// SIMATIC S7-200 project (STEP 7-Micro/WIN), CPU 224XP REL 02.01

SYMBOL_TABLE USUARIO1
P_MOTOR1         I0.0
P_MOTOR2         I0.1
P_PARO           I0.2
MOTOR_1          Q0.0
MOTOR_2          Q0.1
COUNT_SG_M1      VW0      // VARIABLE ENCARGADA DE CONTAR LOS SG DE FUNCIONAMIENTO DEL MOTOR 1
COUNT_MIN_M1     VW2
COUNT_HORS_M1    VD4      // CUENTA LAS HORAS CON UNA DOBLE PALABRA  MAS DE 4000 MILLONES
COUNT_SG_M2      VW8      // VARIABLE ENCARGADA DE CONTAR LOS SG DE FUNCIONAMIENTO DEL MOTOR 1
COUNT_MIN_M2     VW10
COUNT_HORS_M2    VD12     // CUENTA LAS HORAS CON UNA DOBLE PALABRA  MAS DE 4000 MILLONES
COUNT_SG_TOT     VW15     // VARIABLE ENCARGADA DE CONTAR LOS SG DE FUNCIONAMIENTO DEL MOTOR 1
COUNT_MIN_TOT    VW17
COUNT_HORS_TOT   VD20     // HORAS TOTALES
END_SYMBOL_TABLE

SYMBOL_TABLE Símbolos S7-200
Siempre_ON       SM0.0    // Siempre ON
Reloj_1s         SM0.5    // Reloj ON durante 0,5 s, OFF durante 0,5 s, tiempo de ciclo = 1 s.
END_SYMBOL_TABLE

ORGANIZATION_BLOCK PRINCIPAL:OB1
TITLE=CONTADOR HORAS MOTORES
BEGIN
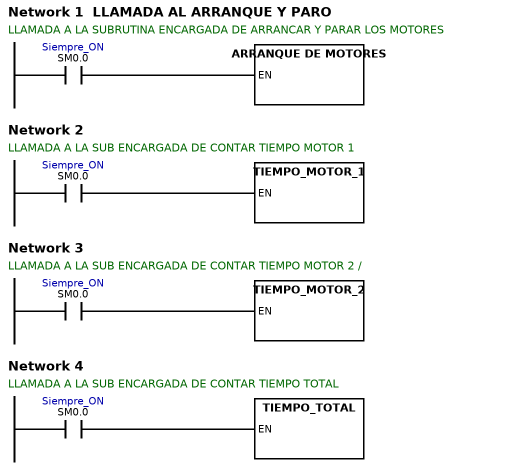
Network 1 // LLAMADA AL ARRANQUE Y PARO
// LLAMADA A LA SUBRUTINA ENCARGADA DE ARRANCAR Y PARAR LOS MOTORES
LD     Siempre_ON:SM0.0
CALL   ARRANQUE DE MOTORES:SBR0
Network 2
// LLAMADA A LA SUB ENCARGADA DE CONTAR TIEMPO MOTOR 1
LD     Siempre_ON:SM0.0
CALL   TIEMPO_MOTOR_1:SBR1
Network 3
// LLAMADA A LA SUB ENCARGADA DE CONTAR TIEMPO MOTOR 2
// 
LD     Siempre_ON:SM0.0
CALL   TIEMPO_MOTOR_2:SBR2
Network 4
// LLAMADA A LA SUB ENCARGADA DE CONTAR TIEMPO TOTAL
LD     Siempre_ON:SM0.0
CALL   TIEMPO_TOTAL:SBR3
END_ORGANIZATION_BLOCK

SUBROUTINE_BLOCK ARRANQUE DE MOTORES:SBR0
TITLE=SUBRUTINA ENCARGADA DE ARRANCAR Y PARAR LOS DOS MOTORES
BEGIN
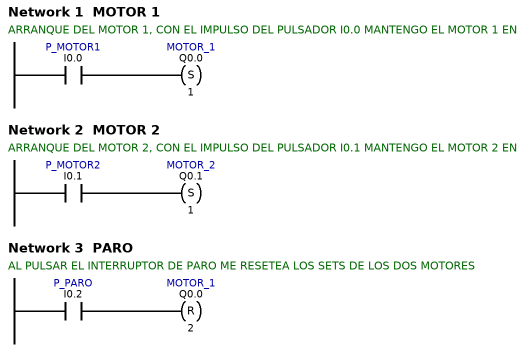
Network 1 // MOTOR 1
// ARRANQUE DEL MOTOR 1, CON EL IMPULSO DEL PULSADOR I0.0 MANTENGO EL MOTOR 1 EN SET
LD     P_MOTOR1:I0.0
S      MOTOR_1:Q0.0, 1
Network 2 // MOTOR 2
// ARRANQUE DEL MOTOR 2, CON EL IMPULSO DEL PULSADOR I0.1 MANTENGO EL MOTOR 2 EN SET
LD     P_MOTOR2:I0.1
S      MOTOR_2:Q0.1, 1
Network 3 // PARO 
// AL PULSAR EL INTERRUPTOR DE PARO ME RESETEA LOS SETS DE LOS DOS MOTORES
LD     P_PARO:I0.2
R      MOTOR_1:Q0.0, 2
END_SUBROUTINE_BLOCK

SUBROUTINE_BLOCK TIEMPO_MOTOR_1:SBR1
TITLE=CONTAJE DEL TIEMPO DEL FUNCIONAMIENTO DEL MOTOR 1
BEGIN
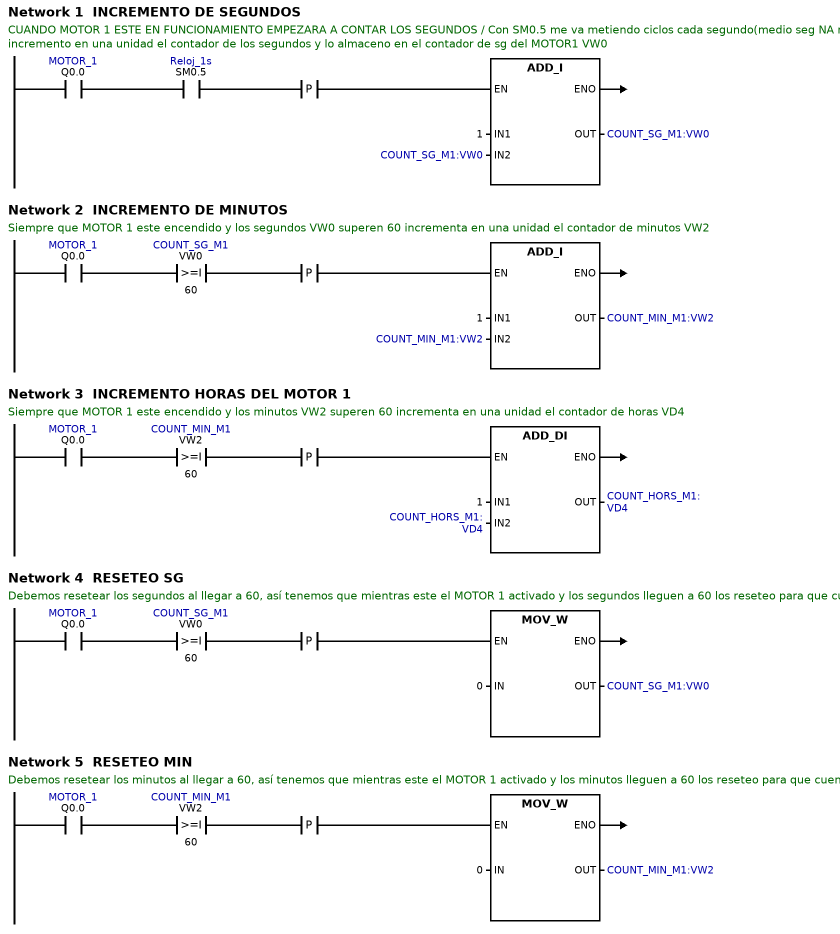
Network 1 // INCREMENTO DE SEGUNDOS
// CUANDO MOTOR 1 ESTE EN FUNCIONAMIENTO EMPEZARA A CONTAR LOS SEGUNDOS
// Con SM0.5 me va metiendo ciclos cada segundo(medio seg NA medio seg nb). Por cada impulso de SM0.5 incremento en una unidad el contador de los segundos y lo almaceno en el contador de sg del MOTOR1 VW0
LD     MOTOR_1:Q0.0
A      Reloj_1s:SM0.5
EU
+I     1, COUNT_SG_M1:VW0
Network 2 // INCREMENTO DE MINUTOS		
// Siempre que MOTOR 1 este encendido y los segundos VW0 superen 60 incrementa en una unidad el contador de minutos VW2
LD     MOTOR_1:Q0.0
AW>=   COUNT_SG_M1:VW0, 60
EU
+I     1, COUNT_MIN_M1:VW2
Network 3 // INCREMENTO HORAS DEL MOTOR 1
// Siempre que MOTOR 1 este encendido y los minutos VW2 superen 60 incrementa en una unidad el contador de horas VD4
LD     MOTOR_1:Q0.0
AW>=   COUNT_MIN_M1:VW2, 60
EU
+D     1, COUNT_HORS_M1:VD4
Network 4 // RESETEO SG
// Debemos resetear los segundos al llegar a 60, así tenemos que mientras este el MOTOR 1 activado y los segundos lleguen a 60 los reseteo para que cuenten el siguiente minuto
LD     MOTOR_1:Q0.0
AW>=   COUNT_SG_M1:VW0, 60
EU
MOVW   0, COUNT_SG_M1:VW0
Network 5 // RESETEO MIN
// Debemos resetear los minutos al llegar a 60, así tenemos que mientras este el MOTOR 1 activado y los minutos lleguen a 60 los reseteo para que cuenten la siguiente hora
LD     MOTOR_1:Q0.0
AW>=   COUNT_MIN_M1:VW2, 60
EU
MOVW   0, COUNT_MIN_M1:VW2
END_SUBROUTINE_BLOCK

SUBROUTINE_BLOCK TIEMPO_MOTOR_2:SBR2
TITLE=CONTAJE DEL TIEMPO DE FUNCIONAMIENTO DEL MOTOR 2
BEGIN
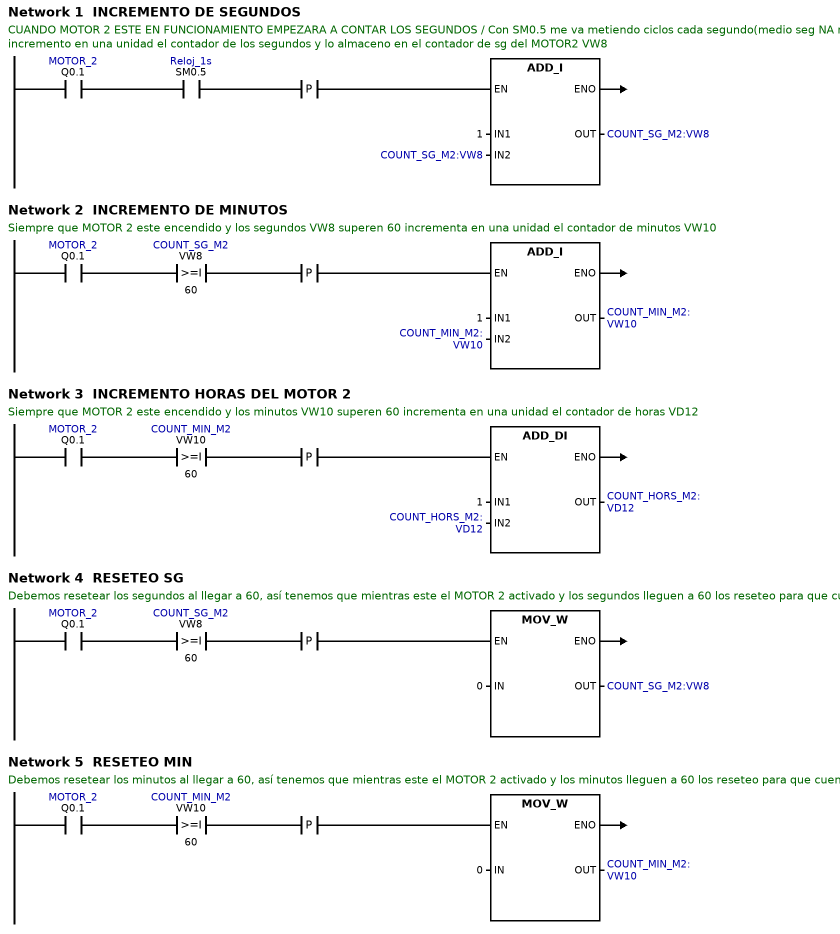
Network 1 // INCREMENTO DE SEGUNDOS
// CUANDO MOTOR 2 ESTE EN FUNCIONAMIENTO EMPEZARA A CONTAR LOS SEGUNDOS
// Con SM0.5 me va metiendo ciclos cada segundo(medio seg NA medio seg nb). Por cada impulso de SM0.5 incremento en una unidad el contador de los segundos y lo almaceno en el contador de sg del MOTOR2 VW8
LD     MOTOR_2:Q0.1
A      Reloj_1s:SM0.5
EU
+I     1, COUNT_SG_M2:VW8
Network 2 // INCREMENTO DE MINUTOS		
// Siempre que MOTOR 2 este encendido y los segundos VW8 superen 60 incrementa en una unidad el contador de minutos VW10
LD     MOTOR_2:Q0.1
AW>=   COUNT_SG_M2:VW8, 60
EU
+I     1, COUNT_MIN_M2:VW10
Network 3 // INCREMENTO HORAS DEL MOTOR 2
// Siempre que MOTOR 2 este encendido y los minutos VW10 superen 60 incrementa en una unidad el contador de horas VD12
LD     MOTOR_2:Q0.1
AW>=   COUNT_MIN_M2:VW10, 60
EU
+D     1, COUNT_HORS_M2:VD12
Network 4 // RESETEO SG
// Debemos resetear los segundos al llegar a 60, así tenemos que mientras este el MOTOR 2 activado y los segundos lleguen a 60 los reseteo para que cuenten el siguiente minuto
LD     MOTOR_2:Q0.1
AW>=   COUNT_SG_M2:VW8, 60
EU
MOVW   0, COUNT_SG_M2:VW8
Network 5 // RESETEO MIN
// Debemos resetear los minutos al llegar a 60, así tenemos que mientras este el MOTOR 2 activado y los minutos lleguen a 60 los reseteo para que cuenten la siguiente hora
LD     MOTOR_2:Q0.1
AW>=   COUNT_MIN_M2:VW10, 60
EU
MOVW   0, COUNT_MIN_M2:VW10
END_SUBROUTINE_BLOCK

SUBROUTINE_BLOCK TIEMPO_TOTAL:SBR3
TITLE=TIEMPO TOTAL INVERTIDO EN LOS DOS MOTORES
BEGIN
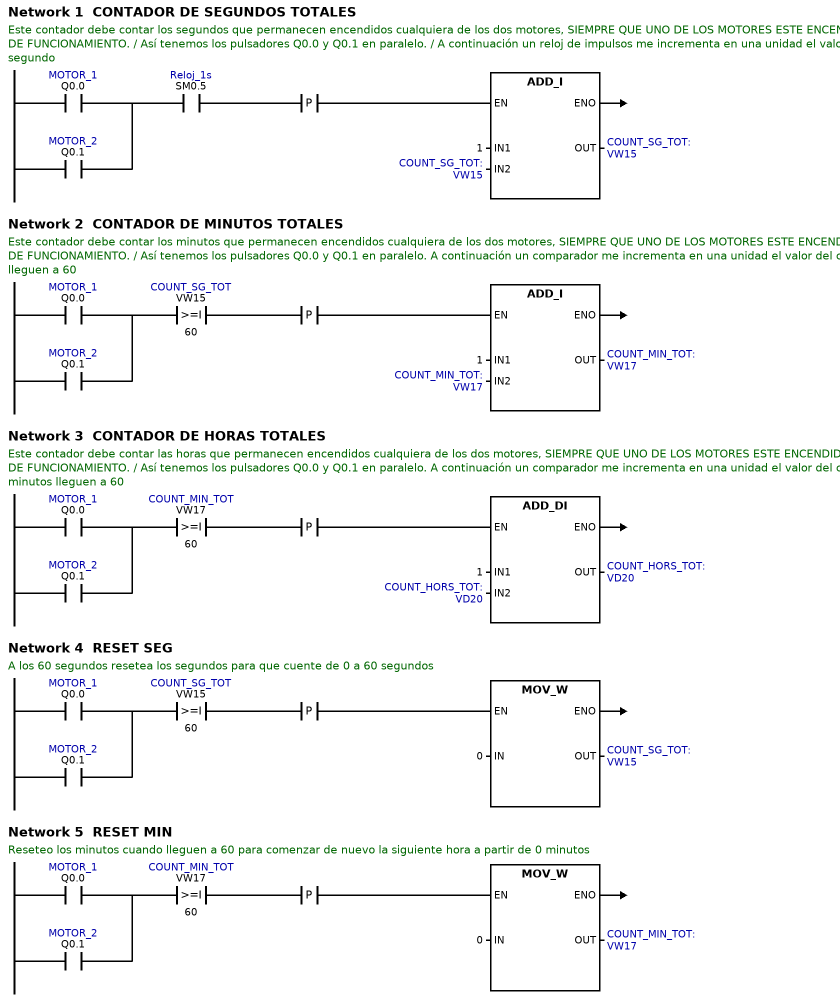
Network 1 // CONTADOR DE SEGUNDOS TOTALES
// Este contador debe contar los segundos que permanecen encendidos cualquiera de los dos motores, SIEMPRE QUE UNO DE LOS MOTORES ESTE ENCENDIDO ESTE CONTADOR DEBE CONTAR LOS SG DE FUNCIONAMIENTO.
// Así tenemos los pulsadores Q0.0 y Q0.1 en paralelo.
// A continuación un reloj de impulsos me incrementa en una unidad el valor del contador de segundos VW15 a cada segundo
LD     MOTOR_1:Q0.0
O      MOTOR_2:Q0.1
A      Reloj_1s:SM0.5
EU
+I     1, COUNT_SG_TOT:VW15
Network 2 // CONTADOR DE MINUTOS TOTALES
// Este contador debe contar los minutos que permanecen encendidos cualquiera de los dos motores, SIEMPRE QUE UNO DE LOS MOTORES ESTE ENCENDIDO ESTE CONTADOR DEBE CONTAR LOS MIN DE FUNCIONAMIENTO.
// Así tenemos los pulsadores Q0.0 y Q0.1 en paralelo. A continuación un comparador me incrementa en una unidad el valor del contador de minutos VW17 cada vez que los sg lleguen a 60
LD     MOTOR_1:Q0.0
O      MOTOR_2:Q0.1
AW>=   COUNT_SG_TOT:VW15, 60
EU
+I     1, COUNT_MIN_TOT:VW17
Network 3 // CONTADOR DE HORAS TOTALES
// Este contador debe contar las horas que permanecen encendidos cualquiera de los dos motores, SIEMPRE QUE UNO DE LOS MOTORES ESTE ENCENDIDO ESTE CONTADOR DEBE CONTAR LAS HORAS DE FUNCIONAMIENTO.
// Así tenemos los pulsadores Q0.0 y Q0.1 en paralelo. A continuación un comparador me incrementa en una unidad el valor del contador de horas VD20 cada vez que los minutos lleguen a 60
LD     MOTOR_1:Q0.0
O      MOTOR_2:Q0.1
AW>=   COUNT_MIN_TOT:VW17, 60
EU
+D     1, COUNT_HORS_TOT:VD20
Network 4 // RESET SEG
// A los 60 segundos resetea los segundos para que cuente de 0 a 60 segundos
LD     MOTOR_1:Q0.0
O      MOTOR_2:Q0.1
AW>=   COUNT_SG_TOT:VW15, 60
EU
MOVW   0, COUNT_SG_TOT:VW15
Network 5 // RESET MIN
// Reseteo los minutos cuando lleguen a 60 para comenzar de nuevo la siguiente hora a partir de 0 minutos
LD     MOTOR_1:Q0.0
O      MOTOR_2:Q0.1
AW>=   COUNT_MIN_TOT:VW17, 60
EU
MOVW   0, COUNT_MIN_TOT:VW17
END_SUBROUTINE_BLOCK
